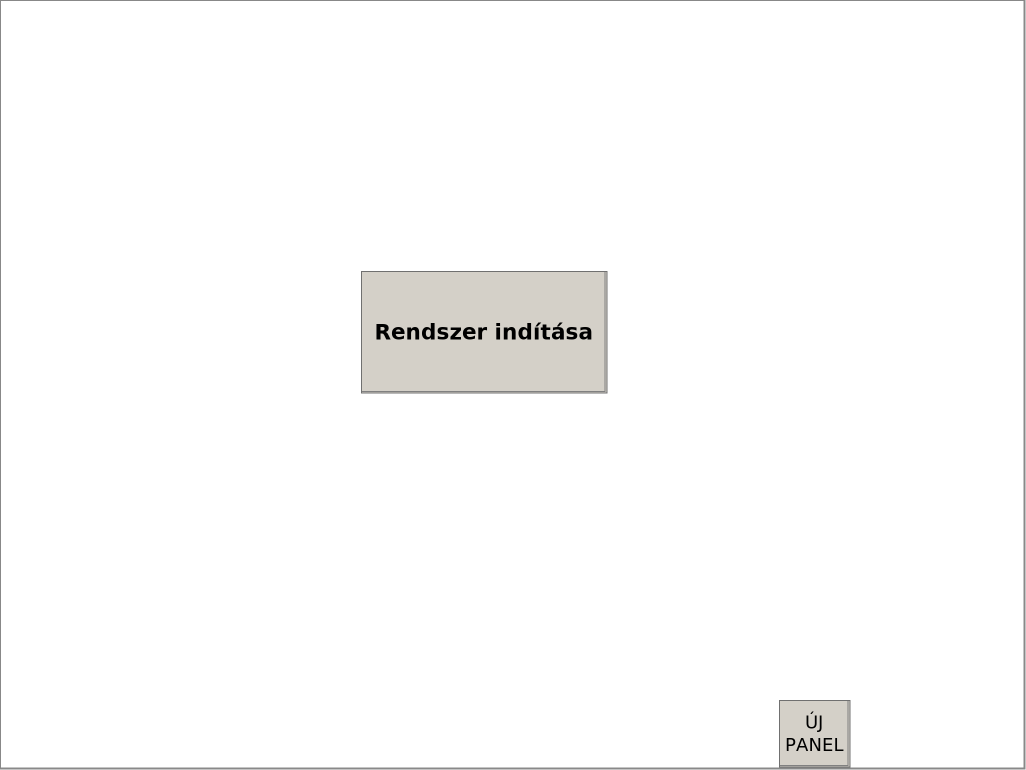
VISUALIZATION Visualization_old  // 1026x770
    TabControl (0,0 1024x768), invisible if: GVL.bSystemNotStarted, input disabled if: GVL.bSystemNotStarted
        shows Termeles()
        shows Termeles1()
        shows Termeles2()
        shows TempZoli()
        shows TempRobot()
        shows TempJozsi()
        shows TempPisti()
        shows Laser()
        shows HegesztesGrafikon()
        [0]: TabTitle=Termelés
        [3]: TabTitle=Főnök
        [4]: TabTitle=Robot
        [5]: TabTitle=Józsi
        [6]: TabTitle=Pisti
        [7]: TabTitle=Lézer
        [8]: TabTitle=Útmérés
    Button (361,271 246x122), "Rendszer indítása", invisible if: GVL.bSystemStarted, input disabled if: GVL.bSystemStarted
        OnMouseClick: execute { INIT.iState:=1; }
    Button (779,700 71x67), "ÚJ PANEL", invisible if: GVL.bSystemNotStarted, input disabled if: GVL.bSystemNotStarted
        OnMouseClick: execute { GVL.bRegiFelulet:=FALSE; }
END_VISUALIZATION

(* stored: Version 1.1.0.1, ProductVersion 3.1.4024.11
   Visu Visualization_old: Id {0aedc4fa-7859-46d0-94f7-778e054ceb42} *)
